(* IEC 61131-3 sources: repolevel_ST_code_completion/output/full_case_fixed/repoeval_four-level_elevator_control/readful_result_history, 9 files *)

(* ---- F_CheckJobInDirection_0.st ---- *)
FUNCTION F_CheckJobInDirection : BOOL
VAR_INPUT
	nStartFloor		:	USINT;		//起始楼层
	nEndFloor		:	USINT;		//结束楼层
	bIncreasing		:	BOOL;		//TRUE=向上检查（递增），FALSE=向下检查（递减）
END_VAR
VAR
	i	:	USINT;
END_VAR

F_CheckJobInDirection := FALSE;

IF bIncreasing THEN
	// 向上检查（从低楼层到高楼层）
	FOR i := nStartFloor TO nEndFloor DO
		IF Tar_Dir.IsStopFloor[i] THEN
			F_CheckJobInDirection := TRUE;
			RETURN;
		END_IF
	END_FOR
ELSE
	// 向下检查（从高楼层到低楼层）
	FOR i := nEndFloor TO nStartFloor BY -1 DO
		IF Tar_Dir.IsStopFloor[i] THEN
			F_CheckJobInDirection := TRUE;
			RETURN;
		END_IF
	END_FOR
END_IF

RETURN;
END_FUNCTION

(* ---- F_CheckJobInDirection_1.st ---- *)
FUNCTION F_CheckJobInDirection : BOOL
VAR_INPUT
	nStartFloor		:	USINT;		//起始楼层
	nEndFloor		:	USINT;		//结束楼层
	bIncreasing		:	BOOL;		//TRUE=向上检查（递增），FALSE=向下检查（递减）
END_VAR
VAR
	i	:	USINT;
END_VAR

F_CheckJobInDirection := FALSE;

IF bIncreasing THEN
	// 向上检查（从低楼层到高楼层）
	FOR i := nStartFloor TO nEndFloor DO
		IF Tar_Dir.IsStopFloor[i] THEN
			F_CheckJobInDirection := TRUE;
			RETURN;
		END_IF
	END_FOR
ELSE
	// 向下检查（从高楼层到低楼层）
i := nEndFloor; // Initialize i to nEndFloor
  WHILE i >= nStartFloor DO
    IF Tar_Dir.IsStopFloor[i] THEN
      F_CheckJobInDirection := TRUE;
      RETURN;
    END_IF
    i := i - 1; // Decrement i manually to avoid using BY -1 with USINT
  END_WHILE
END_IF

RETURN;
END_FUNCTION

(* ---- F_CheckJobInDirection_2.st ---- *)
FUNCTION F_CheckJobInDirection : BOOL
VAR_INPUT
	nStartFloor		:	USINT;		//起始楼层
	nEndFloor		:	USINT;		//结束楼层
	bIncreasing		:	BOOL;		//TRUE=向上检查（递增），FALSE=向下检查（递减）
END_VAR
VAR
	i	:	USINT;
END_VAR

F_CheckJobInDirection := FALSE;

IF bIncreasing THEN
	// 向上检查（从低楼层到高楼层）
	FOR i := nStartFloor TO nEndFloor DO
		IF Tar_Dir.IsStopFloor[i] THEN
			F_CheckJobInDirection := TRUE;
			RETURN;
		END_IF
	END_FOR
ELSE
	// 向下检查（从高楼层到低楼层）
i := nEndFloor; // Initialize i to nEndFloor
 WHILE i >= nStartFloor AND i <= 255 DO // Add explicit bounds check for USINT range (0 to 255)
  IF Tar_Dir.IsStopFloor[i] THEN
   F_CheckJobInDirection := TRUE;
   RETURN;
  END_IF
  IF i > 0 THEN  // Ensure i does not become less than zero
   i := i - 1; // Decrement within valid USINT range
  ELSE
   EXIT; // Stop the loop if i reaches 0, preventing underflow
  END_IF
 END_WHILE
END_IF

RETURN;
END_FUNCTION

(* ---- F_CheckJobInDirection_3.st ---- *)
FUNCTION F_CheckJobInDirection : BOOL
VAR_INPUT
	nStartFloor		:	USINT;		//起始楼层
	nEndFloor		:	USINT;		//结束楼层
	bIncreasing		:	BOOL;		//TRUE=向上检查（递增），FALSE=向下检查（递减）
END_VAR
VAR
	i	:	USINT;
END_VAR

F_CheckJobInDirection := FALSE;

IF bIncreasing THEN
	// 向上检查（从低楼层到高楼层）
	FOR i := nStartFloor TO nEndFloor DO
		IF Tar_Dir.IsStopFloor[i] THEN
			F_CheckJobInDirection := TRUE;
			RETURN;
		END_IF
	END_FOR
ELSE
	// 向下检查（从高楼层到低楼层）
i := nEndFloor; // Initialize i to nEndFloor
WHILE i >= nStartFloor DO // Simplify logic by removing unnecessary bounds check; `USINT` naturally limits to 255
 IF Tar_Dir.IsStopFloor[i] THEN
  F_CheckJobInDirection := TRUE;
  RETURN;
 END_IF
 IF i = 0 THEN // Check explicitly for underflow
  EXIT; // Exit the loop if `i` reaches its lower bound (0)
 ELSE
  i := i - 1; // Decrement safely within valid range
 END_IF
END_WHILE
END_IF

RETURN;
END_FUNCTION

(* ---- F_ClearFloorStop_0.st ---- *)
FUNCTION F_ClearFloorStop
VAR_INPUT
	nFloor			:	USINT;		//楼层号
	bClearUpStop	:	BOOL;		//是否清除上升停靠标志
	bClearDownStop	:	BOOL;		//是否清除下降停靠标志
	bClearStopFloor	:	BOOL;		//是否清除楼层停靠标志
END_VAR
IF bClearUpStop AND (nFloor <= MaxNumFloor - 1) THEN
	Tar_Dir.IsUpStop[nFloor] := FALSE;
	QFloorUpLed[nFloor] := FALSE;
END_IF;

IF bClearDownStop AND (nFloor >= 2) THEN
	Tar_Dir.IsDownStop[nFloor] := FALSE;
	QFloorDownLed[nFloor] := FALSE;
END_IF;

IF bClearStopFloor THEN
	Tar_Dir.IsStopFloor[nFloor] := FALSE;
	QGoFloorLed[nFloor] := FALSE;
END_IF;

RETURN;
END_FUNCTION

(* ---- F_ClearFloorStop_1.st ---- *)
FUNCTION F_ClearFloorStop
VAR_INPUT
  nFloor			:	USINT;		//楼层号
  bClearUpStop	:	BOOL;		//是否清除上升停靠标志
  bClearDownStop	:	BOOL;		//是否清除下降停靠标志
  bClearStopFloor	:	BOOL;		//是否清除楼层停靠标志
END_VAR
IF bClearUpStop AND (nFloor <= MaxNumFloor - 1) THEN
  IF nFloor >= 1 THEN // Ensure that nFloor is within valid bounds for the IsUpStop array
    Tar_Dir.IsUpStop[nFloor] := FALSE;
    QFloorUpLed[nFloor] := FALSE;
  END_IF;
END_IF;

IF bClearDownStop AND (nFloor >= 2) THEN
  IF nFloor <= MaxNumFloor THEN // Check bounds for IsDownStop array
    Tar_Dir.IsDownStop[nFloor] := FALSE;
    QFloorDownLed[nFloor] := FALSE;
  END_IF;
END_IF;

IF bClearStopFloor THEN
  IF nFloor >= 1 AND nFloor <= MaxNumFloor THEN // Ensure nFloor is a valid index for IsStopFloor array
    Tar_Dir.IsStopFloor[nFloor] := FALSE;
    QGoFloorLed[nFloor] := FALSE;
  END_IF;
END_IF;

RETURN;
END_FUNCTION

(* ---- F_ClearFloorStop_2.st ---- *)
FUNCTION F_ClearFloorStop
VAR_INPUT
 nFloor			:	USINT;		//楼层号
 bClearUpStop	:	BOOL;		//是否清除上升停靠标志
 bClearDownStop	:	BOOL;		//是否清除下降停靠标志
 bClearStopFloor	:	BOOL;		//是否清除楼层停靠标志
END_VAR
// Assuming a known fixed limit for the number of floors, replace MaxNumFloor with an explicit value (e.g., 10).
IF bClearUpStop AND (nFloor <= 9) THEN // Substitute MaxNumFloor - 1 with 9
 IF nFloor >= 1 THEN // Ensure that nFloor is within valid bounds for the IsUpStop array
  Tar_Dir.IsUpStop[nFloor] := FALSE;
  QFloorUpLed[nFloor] := FALSE;
 END_IF;
END_IF;

IF bClearDownStop AND (nFloor >= 2) THEN
 IF nFloor <= 10 THEN // Substitute MaxNumFloor with 10
  Tar_Dir.IsDownStop[nFloor] := FALSE;
  QFloorDownLed[nFloor] := FALSE;
 END_IF;
END_IF;

IF bClearStopFloor THEN
 IF nFloor >= 1 AND nFloor <= 10 THEN // Substitute MaxNumFloor with 10
  Tar_Dir.IsStopFloor[nFloor] := FALSE;
  QGoFloorLed[nFloor] := FALSE;
 END_IF;
END_IF;

RETURN;
END_FUNCTION

(* ---- F_ClearFloorStop_3.st ---- *)
FUNCTION F_ClearFloorStop
VAR_INPUT
nFloor			:	USINT;		//楼层号
bClearUpStop	:	BOOL;		//是否清除上升停靠标志
bClearDownStop	:	BOOL;		//是否清除下降停靠标志
bClearStopFloor	:	BOOL;		//是否清除楼层停靠标志
END_VAR
// Simplified and combined boundary checks to improve clarity and avoid redundancy
IF bClearUpStop AND (nFloor >= 1 AND nFloor <= 9) THEN
 Tar_Dir.IsUpStop[nFloor] := FALSE;
 QFloorUpLed[nFloor] := FALSE;
END_IF;

IF bClearDownStop AND (nFloor >= 2 AND nFloor <= 10) THEN
 Tar_Dir.IsDownStop[nFloor] := FALSE;
 QFloorDownLed[nFloor] := FALSE;
END_IF;

IF bClearStopFloor AND (nFloor >= 1 AND nFloor <= 10) THEN
 Tar_Dir.IsStopFloor[nFloor] := FALSE;
 QGoFloorLed[nFloor] := FALSE;
END_IF;

RETURN;
END_FUNCTION

(* ---- F_SetElevatorDirection_0.st ---- *)
FUNCTION F_SetElevatorDirection
VAR_INPUT
	nCurrentFloor	:	USINT;		//当前楼层
	nTargetFloor	:	USINT;		//目标楼层
END_VAR
VAR
	bDirectionSet   :   BOOL;       //标志是否已设置方向
END_VAR

bDirectionSet := FALSE;

// 根据当前楼层和目标楼层设定电梯运行方向
IF nTargetFloor > nCurrentFloor THEN
	// 目标楼层高于当前楼层，电梯上升
	Tar_Dir.IsPositive := TRUE;
	Tar_Dir.IsNegative := FALSE;
	bDirectionSet := TRUE;
ELSIF nTargetFloor < nCurrentFloor THEN
	// 目标楼层低于当前楼层，电梯下降
	Tar_Dir.IsPositive := FALSE;
	Tar_Dir.IsNegative := TRUE;
	bDirectionSet := TRUE;
END_IF;

// 如果目标楼层等于当前楼层，不改变方向
IF NOT bDirectionSet THEN
	Tar_Dir.IsPositive := FALSE;
	Tar_Dir.IsNegative := FALSE;
END_IF;

RETURN;
END_FUNCTION
